_CFC_ (* Continuous Function Chart, elements in execution order *)
(* 85% от частоты вращения *)
(* 60% от частоты вращения *)
#0 WORD_TO_REAL(RD_2[0])
#1 DIV(#0, 100)
#2 SHU6_PV1_MV1_OBR <= #1
#3 dost_ton_3:TON(IN: NOT SHU6_PV1_MV1_OBR_ERROR, PT: t#10s)
#4 SR_DOST_MV1:RS(SET: #3.Q, RESET1: SHU6_PV1_MV1_OBR_ERROR)
#5 DIV(SHU6_PV1_M_MAXSPEED, 100)
#6 MUL(#5, 60)
#7 fb_MV1b30:ISTOK_GT(dost: #4.Q1, x: SHU6_PV1_MV1_OBR, ust: #6, shkal: -, gist: 1)
#8 SHU6_PV1_MV1_B30 <= #7.Xb
#9 DIV(SHU6_PV1_M_MAXSPEED, 100)
#10 MUL(#9, 85)
#11 fb_MV1_OBRb45:ISTOK_GT(dost: #4.Q1, x: SHU6_PV1_MV1_OBR, ust: #10, shkal: -, gist: 1)
#12 SHU6_PV1_MV1_B45 <= #11.Xb
#13 fb_MV1_OBRm0_1:ISTOK_LT(dost: #4.Q1, x: SHU6_PV1_MV1_OBR, ust: 0.1, shkal: -, gist: 1)
#14 SHU6_PV1_MV1_M0_1 <= #13.Xm
#15 fb_MV1_OBRbSM:ISTOK_GT(dost: #4.Q1, x: SHU6_PV1_MV1_OBR, ust: SHU6_PV1_M_MAXSPEED, shkal: -, gist: 1)
#16 SHU6_PV1_MV1_OBRBSM <= #15.Xb
_END_CFC_
(* the same logic as Structured Text *)
(* 85% от частоты вращения *)
(* 60% от частоты вращения *)
SHU6_PV1_MV1_OBR := WORD_TO_REAL(RD_2[0]) / 100;
dost_ton_3(IN := NOT SHU6_PV1_MV1_OBR_ERROR, PT := t#10s);
SR_DOST_MV1(SET := dost_ton_3.Q, RESET1 := SHU6_PV1_MV1_OBR_ERROR);
fb_MV1b30(dost := SR_DOST_MV1.Q1, x := SHU6_PV1_MV1_OBR, ust := (SHU6_PV1_M_MAXSPEED / 100) * 60, gist := 1);
SHU6_PV1_MV1_B30 := fb_MV1b30.Xb;
fb_MV1_OBRb45(dost := SR_DOST_MV1.Q1, x := SHU6_PV1_MV1_OBR, ust := (SHU6_PV1_M_MAXSPEED / 100) * 85, gist := 1);
SHU6_PV1_MV1_B45 := fb_MV1_OBRb45.Xb;
fb_MV1_OBRm0_1(dost := SR_DOST_MV1.Q1, x := SHU6_PV1_MV1_OBR, ust := 0.1, gist := 1);
SHU6_PV1_MV1_M0_1 := fb_MV1_OBRm0_1.Xm;
fb_MV1_OBRbSM(dost := SR_DOST_MV1.Q1, x := SHU6_PV1_MV1_OBR, ust := SHU6_PV1_M_MAXSPEED, gist := 1);
SHU6_PV1_MV1_OBRBSM := fb_MV1_OBRbSM.Xb;
END_PROGRAM

(* POU Input/AI/TE6, CFC *)
PROGRAM TE6
VAR
	fb_UE2_T: ISTOK_ANALOGVH;
	ofset: REAL;
	fb_UE2eqUST: ISTOK_EQ;
	enbleLimit: BOOL;
	fb_TE6_m_UST: ISTOK_LT;
	fb_TE6_b_UST: ISTOK_GT;
	I_GT_TE: ISTOK_GT;
	I_LT_TE: ISTOK_LT;
	TON_DOST: TON;
END_VAR
VAR (* helpers for the ST form of the networks *)
	_t76 : REAL;
END_VAR
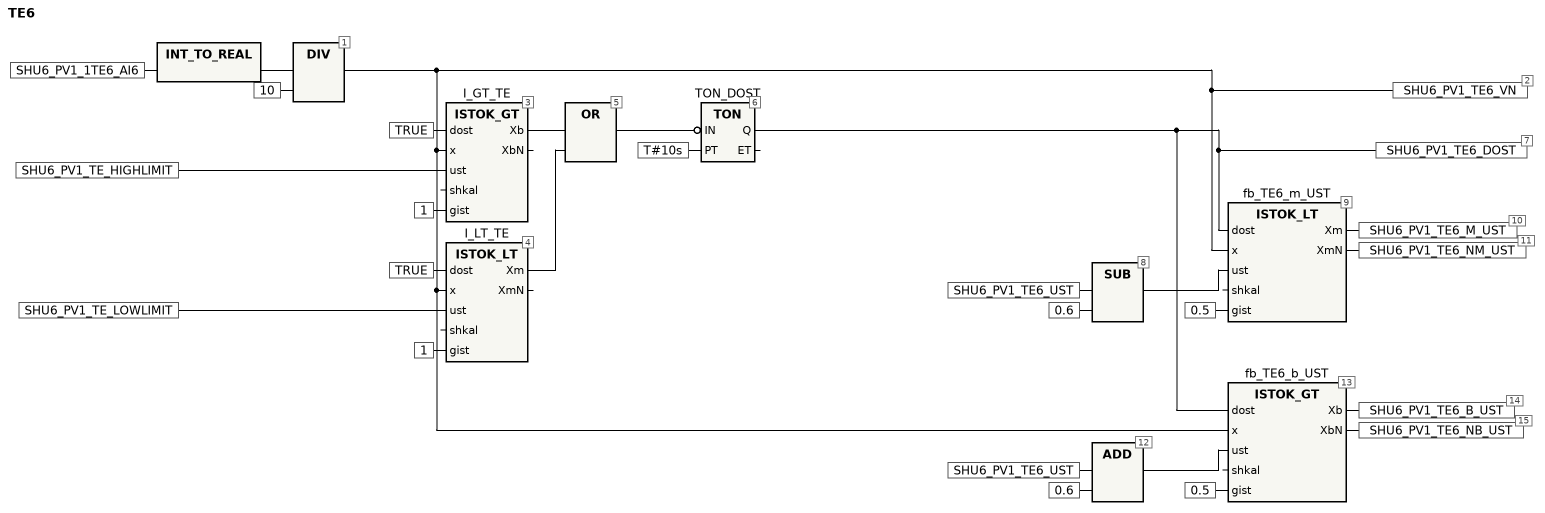
_CFC_ (* Continuous Function Chart, elements in execution order *)
#0 INT_TO_REAL(SHU6_PV1_1TE6_AI6)
#1 DIV(#0, 10)
#2 SHU6_PV1_TE6_VN <= #1
#3 I_GT_TE:ISTOK_GT(dost: TRUE, x: #1, ust: SHU6_PV1_TE_HIGHLIMIT, shkal: -, gist: 1)
#4 I_LT_TE:ISTOK_LT(dost: TRUE, x: #1, ust: SHU6_PV1_TE_LOWLIMIT, shkal: -, gist: 1)
#5 OR(#3.Xb, #4.Xm)
#6 TON_DOST:TON(IN: NOT #5, PT: T#10s)
#7 SHU6_PV1_TE6_DOST <= #6.Q
#8 SUB(SHU6_PV1_TE6_UST, 0.6)
#9 fb_TE6_m_UST:ISTOK_LT(dost: #6.Q, x: #1, ust: #8, shkal: -, gist: 0.5)
#10 SHU6_PV1_TE6_M_UST <= #9.Xm
#11 SHU6_PV1_TE6_NM_UST <= #9.XmN
#12 ADD(SHU6_PV1_TE6_UST, 0.6)
#13 fb_TE6_b_UST:ISTOK_GT(dost: #6.Q, x: #1, ust: #12, shkal: -, gist: 0.5)
#14 SHU6_PV1_TE6_B_UST <= #13.Xb
#15 SHU6_PV1_TE6_NB_UST <= #13.XbN
_END_CFC_
(* the same logic as Structured Text *)
_t76 := INT_TO_REAL(SHU6_PV1_1TE6_AI6) / 10;
SHU6_PV1_TE6_VN := _t76;
I_GT_TE(dost := TRUE, x := _t76, ust := SHU6_PV1_TE_HIGHLIMIT, gist := 1);
I_LT_TE(dost := TRUE, x := _t76, ust := SHU6_PV1_TE_LOWLIMIT, gist := 1);
TON_DOST(IN := NOT (I_GT_TE.Xb OR I_LT_TE.Xm), PT := T#10s);
SHU6_PV1_TE6_DOST := TON_DOST.Q;
fb_TE6_m_UST(dost := TON_DOST.Q, x := _t76, ust := SHU6_PV1_TE6_UST - 0.6, gist := 0.5);
SHU6_PV1_TE6_M_UST := fb_TE6_m_UST.Xm;
SHU6_PV1_TE6_NM_UST := fb_TE6_m_UST.XmN;
fb_TE6_b_UST(dost := TON_DOST.Q, x := _t76, ust := SHU6_PV1_TE6_UST + 0.6, gist := 0.5);
SHU6_PV1_TE6_B_UST := fb_TE6_b_UST.Xb;
SHU6_PV1_TE6_NB_UST := fb_TE6_b_UST.XbN;
END_PROGRAM

(* POU Lib/ISTOK_EQ, CFC *)
FUNCTION_BLOCK ISTOK_EQ
VAR_INPUT
	dost: BOOL;
	X: REAL;
	ust: REAL;
	shkal: REAL;
	gist: REAL;
END_VAR
VAR_OUTPUT
	Xeq: BOOL;
	Xneq: BOOL;
END_VAR
VAR
END_VAR
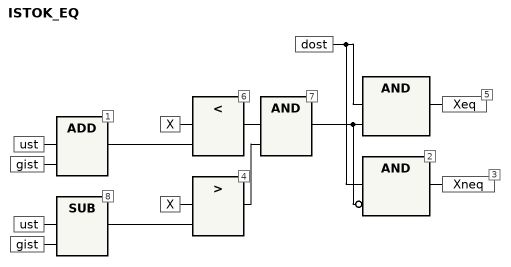
_CFC_ (* Continuous Function Chart, elements in execution order *)
#0 AND(dost, #7)
#1 ADD(ust, gist)
#2 AND(dost, NOT #7)
#3 Xneq <= #2
#4 >(X, #8)
#5 Xeq <= #0
#6 <(X, #1)
#7 AND(#6, #4)
#8 SUB(ust, gist)
_END_CFC_
END_FUNCTION_BLOCK

(* POU Input/AI/TE3, CFC *)
PROGRAM TE3
VAR
	TE3_YST: REAL;
	fb_TE3: ISTOK_ANALOGVH;
	ofset: REAL;
	fb_SHU6_PV1_TE_M_ZASCH: ISTOK_LT;
	fb_SHU6_PV1_TE_M_UST: ISTOK_LT;
	I_GT_TE: ISTOK_GT;
	I_LT_TE: ISTOK_LT;
	TON_DOST: TON;
	SHU6_PV1_TE3_UST: BOOL;
	fb_SHU6_PV1_TE3_M_ZASCH: ISTOK_LT;
	fb_SHU6_PV1_TE3_M_UST: ISTOK_LT;
	fb_TE3_B_UST: ISTOK_GT;
	fb_TE3_M_UST: ISTOK_LT;
END_VAR
VAR (* helpers for the ST form of the networks *)
	_t47 : REAL;
END_VAR
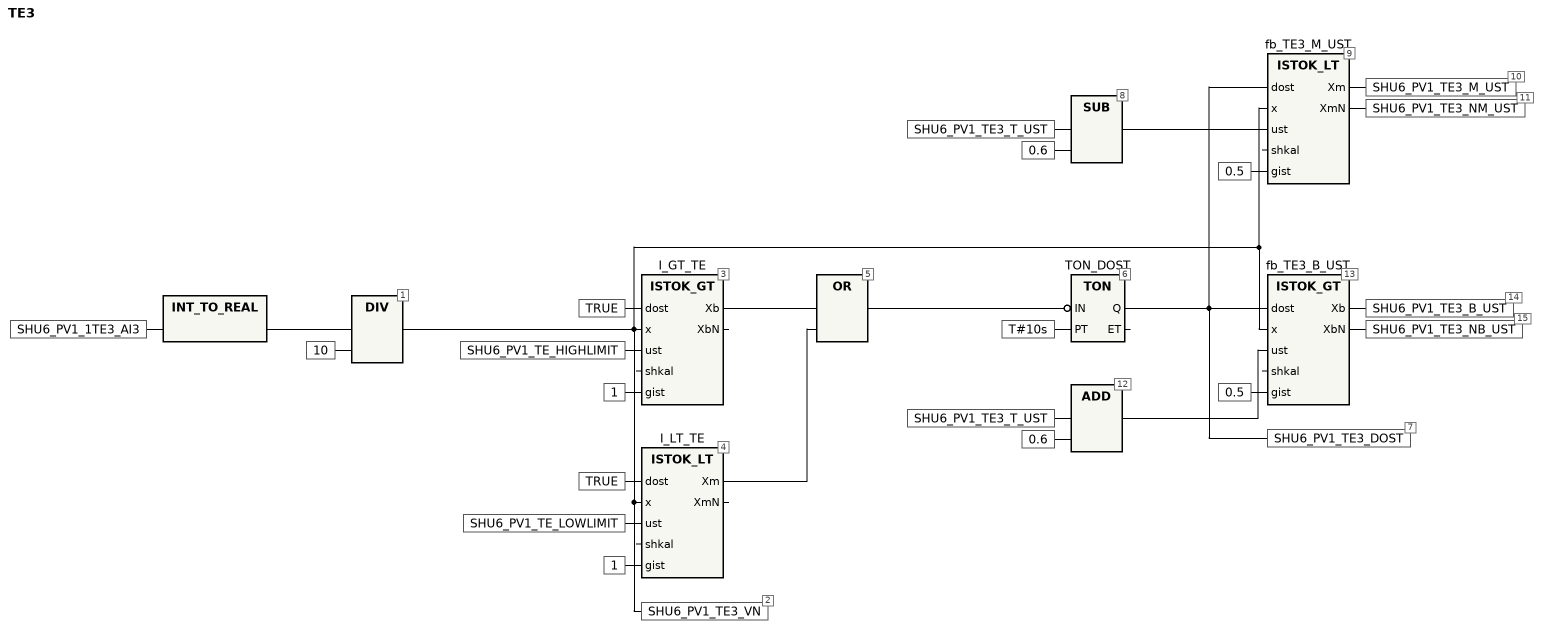
